Staubli VAL3: sampleChangerv5.dtx

bool moveIsStopped
dio switchGripper = {link=valve1}
jointRx binPosition = {j1=59.154914, j2=15.287075, j3=144.068937, j4=0.00349, j5=20.640131, j6=239.148927}
jointRx currentSamPosJ = {j1=64.5166, j2=21.7725, j3=135.395, j4=0.005, j5=22.8226, j6=244.506}
jointRx currentSpinPosJ
jointRx gatePosition = {j1=53.332436, j2=31.008098, j3=108.023775, j4=-0.035914, j5=40.963114, j6=323.353672}
jointRx homePosition = {j1=64.5166, j2=21.7725, j3=135.395, j4=0.005, j5=22.8226, j6=244.506}
jointRx knownPositions{}
  [currentSamPos] = {}
  [currentSpinPos] = {}
  [gatePosition] = {}
  [homePosition] = {}
  [parkingPosition] = {}
  [spinnerHomePos] = {}
  [zeroPosition] = {}
  [binPosition] = {}
jointRx parkingPosition = {j1=20.774519, j2=86.925335, j3=58.285959, j4=-72.455135, j5=101.349332, j6=295.989419}
jointRx spinnerHomePos = {j1=24.038951, j2=102.353577, j3=38.089715, j4=-71.031763, j5=105.005317, j6=322.961782}
jointRx zeroPosition = {j1=88.745927, j2=-26.51301, j3=117.695598, j4=-0.539561, j5=89.308877, j6=269.442332}
mdesc mFastMov = {blend=off}
mdesc mNomSpeed = {accel=2.25, vel=15, decel=2.25}
num numSamOffs[2]
num numSpinOffs[6]
sio sioASCII[2]
  [0] = {link=Socket\tan}
  [1] = {link=Socket\tan}
bool mounted
string calibInfo
